// TIA Portal V17 program export: 0 tag tables, 0 data types, 0 data blocks, 3 code blocks (in call order from the OBs), 0 instance data blocks

ORGANIZATION_BLOCK "Main"   // OB1, LAD, ProgramCycle
TITLE = "Main Program Sweep (Cycle)"
{ S7_Optimized_Access := 'TRUE' }
VERSION : 0.1
// stored: AutoNumber true, IsIECCheckEnabled false, SetENOAutomatically false
   VAR_INPUT
      Initial_Call : Bool;   // Initial call of this OB
      Remanence : Bool;   // =True, if remanent data are available
   END_VAR
   VAR_TEMP   // added for the SCL form of the ladder/FBD networks
      _w1 : Bool;
   END_VAR
BEGIN

REGION Network 1
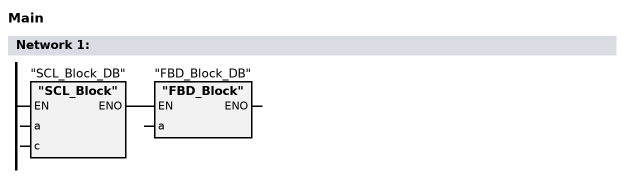
   RUNG wire#powerrail
      "SCL_Block_DB"("a" :=, c :=)
      "FBD_Block_DB"("a" :=)
   END_RUNG
   // the same network as SCL:
   "SCL_Block_DB"(ENO => #_w1);   // "SCL_Block"
   IF #_w1 THEN
       "FBD_Block_DB"();   // "FBD_Block"
   END_IF;
END_REGION
END_ORGANIZATION_BLOCK

FUNCTION_BLOCK "SCL_Block"
{ S7_Optimized_Access := 'TRUE' }
VERSION : 0.1
   VAR_INPUT 
      a : Int;
      c : Int;
   END_VAR

   VAR 
      statCondition : Bool;
   END_VAR


BEGIN
	IF #statCondition = TRUE THEN
	    // Statement section IF
	    
	    ;
	END_IF;
	
	CASE #a OF
	    1:  // Statement section case 1
	        ;
	    2..4:  // Statement section case 2 to 4
	        ;
	    ELSE  // Statement section ELSE
	        ;
	END_CASE;
	
END_FUNCTION_BLOCK

FUNCTION_BLOCK "FBD_Block"   // FB2, FBD
{ S7_Optimized_Access := 'TRUE' }
VERSION : 0.1
// stored: AutoNumber true, IsIECCheckEnabled false, IsRetainMemResEnabled false, MemoryReserve 100, SetENOAutomatically false, UDAEnableTagReadback false
   VAR_INPUT
      "a" : Bool;
   END_VAR
   VAR
      statInfo : Word := 16#5;
      statInfo2 : Word;
   END_VAR
BEGIN

REGION Network 1
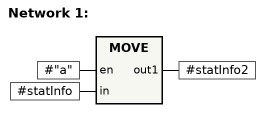
   IF #"a" THEN #statInfo2 := #statInfo; END_IF;
END_REGION
END_FUNCTION_BLOCK
